// TIA Portal V17 export
// export: Created 2025-03-05T08:02:24.076787Z, ExportSetting WithDefaults, DisplayName Totally Integrated Automation Portal, DisplayVersion V17 Update 8, DisplayName TIA Portal Openness, DisplayVersion V17 Update 8, DisplayName TIA Portal Version Control Interface, DisplayVersion V17, DisplayName SINAMICS Startdrive Advanced, DisplayVersion V17 SP2, DisplayName SINAMICS Startdrive G110M, G120, G120C, G120D, G120P, G115D, DisplayVersion V17 SP2, DisplayName SINAMICS Startdrive G130, G150, S120, S150, SINAMICS MV, S210, DisplayVersion V17 SP2, DisplayName STEP 7 Professional, DisplayVersion V17 Update 8, DisplayName SINUMERIK ONE STEP 7 Toolbox, DisplayVersion V17 Update 12, DisplayName SINUMERIK 840D sl STEP 7 Toolbox, DisplayVersion V17 Update 12, DisplayName STEP 7 Safety, DisplayVersion V17 Update 6, DisplayName WinCC Advanced, DisplayVersion V17 Update 8
TYPE "TOOL_LIFE_PLC"
// stored: IsFailsafeCompliant false
   STRUCT
      IS_ALARMS : Bool;   // IMMEDIATE STOP ALARMS
      IS_SEOC_ALARMS : Bool;   // IMMEDIATE STOP & STOP END OF CYCLE ALARMS / IMMEDIATE STOP AND STOP END OF CYCLE ALARMS
      RHP_ALARMS : Bool;   // RETURN HOME POSITION ALARMS
      RHP_SEOC_ALARMS : Bool;   // RETURN HOME POSITION & STOP END OF CYCLE ALARMS / RETURN HOME POSITION AND STOP END OF CYCLE ALARMS
      SEOC_ALARMS : Bool;   // STOP END OF CYCLE ALARMS
      IS_WARNING : Bool;   // IMMEDIATE STOP WARNING / IMMEDIATE STOP WARNINGS
      RHP_WARNING : Bool;   // RETURN HOME POSITION WARNING / RETURN HOME POSITION WARNINGS
      SEOC_WARNING : Bool;   // STOP END OF CYCLE WARNING / STOP END OF CYCLE WARNINGS
      WARNING : Bool;   // WARNING / WARNINGS
      HELP : Bool;   // HELP
      SPARE_11 : Bool;
      SPARE_12 : Bool;
      TOOL_PREALARM : Bool;   // TOOL PREALARM
      TOOL_ALARM : Bool;   // TOOL ALARM
      WARNING_GONE : Bool;   // WARNING GONE
      SPARE_16 : Bool;
      LIFE_EXPIRED_TOOL : Array[1..15] of Bool;   // LIFE EXPIRED TOOL
      SPARE_18 : Bool;
      SPARE_19 : Bool;
      LIFE_WARNING_TOOL : Array[1..15] of Bool;   // LIFE WARNING TOOL
      SPARE_21 : Bool;
      SPARE_22 : Bool;
      COUNTING_ENABLE : Bool;   // COUNTING ENABLE
      COUNTIN_ENABLE_PULSE : Bool;   // COUNTING ENABLE PULSE
      SPARE_25 : Bool;
      SPARE_26 : Bool;
      SPARE_27 : Bool;
      SPARE_28 : Bool;
      SPARE_29 : Bool;
      SPARE_30 : Bool;
   END_STRUCT;
END_TYPE
